(* CODESYS project testPulse_Encoder.project

Project tree, tasks and I/O mapping:
  Device : Jinan Cherry-ARM Cortex-VxWorks, Jinan Cheery Electric Co., Ltd., version 3.5.11.20
    application Application
      libraries: Standard, * (System); CmpModbusLib, 1.0.0 (Hitech); CmpPulseOutput, 1.0.0 (HiTech); CmpGlodonDemo, 1.0.0.0 (Glodon); CmpEncoderCtrl, 1.0.0 (HiTech)
      task MainTask (cyclic, interval 4 ms, priority 1) calls CtrlPulse
      task Encoder (cyclic, interval 500 ms, priority 1) calls ReadEncoder
      program CtrlPulse [ST]
      program ReadEncoder [ST]
    SoftMotion General Axis Pool
*)

// Device/Application/CtrlPulse
PROGRAM CtrlPulse
VAR
	InitOK : BOOL := FALSE;
	isOver : BOOL;
	amount : DWORD := 0;
	SetPulseAmountAndStart : CmpPulseOutput.SetPulseAmountAndStart;
	SetPulseFreq 		   : CmpPulseOutput.SetPulseFreq;
	IsPulseOver 		   : CmpPulseOutput.IsPulseOver;
	StopPulse			   : CmpPulseOutput.StopPulse;
END_VAR

IF InitOk = FALSE THEN
	StopPulse();
	SetPulseFreq(freq:= 10000);
	InitOk := TRUE;
ELSE
	IsPulseOver(isOver=> isOver);
	IF isOver = TRUE AND amount > 0 THEN
		SetPulseAmountAndStart(amount:= amount);
		amount := 0;
	END_IF
END_IF

END_PROGRAM

// Device/Application/ReadEncoder
PROGRAM ReadEncoder
VAR
	InitOK : BOOL := FALSE;

	Direction : BOOL;
	CounterA : DINT;
	CounterZ : DINT;
	ReadEncoderCounterA : CmpEncoderCtrl.ReadEncoderCounterA;
	ReadEncoderCounterZ : CmpEncoderCtrl.ReadEncoderCounterZ;
	ReadEncoderDirection : CmpEncoderCtrl.ReadEncoderDirection;
	SetEncoderCounter : CmpEncoderCtrl.SetEncoderCounter;
END_VAR

IF InitOk = FALSE THEN
	SetEncoderCounter(CounterA:= 0, CounterZ:= 0);
	InitOk := TRUE;
ELSE
	ReadEncoderDirection(Direction=> Direction);
	ReadEncoderCounterA(CounterA=> CounterA);
	ReadEncoderCounterZ(CounterZ=> CounterZ);	
END_IF

END_PROGRAM
